(* IEC 61131-3 sources: PLC-Extruder-project/plc/twincat, 11 files *)

(* ---- DUT_ControllerState.st ---- *)
{attribute 'qualified_only'}
{attribute 'strict'}
TYPE E_ControllerState_Tc :
(
    IDLE := 0,
    STARTUP := 10,
    RUNNING := 20,
    SHUTDOWN := 30,
    EMERGENCY_STOP := 40
);
END_TYPE

(* ---- DUT_ExtruderApp.st ---- *)
{attribute 'qualified_only'}
{attribute 'strict'}
TYPE E_ExtruderMode_Tc :
(
    OFF := 0,
    MANUAL := 10,
    AUTO := 20,
    MAINTENANCE := 30
);
END_TYPE

{attribute 'qualified_only'}
{attribute 'strict'}
TYPE E_RecipeId_Tc :
(
    DEFAULT := 0,
    HDPE_PIPE := 10,
    PVC_PROFILE := 20,
    CUSTOM := 100
);
END_TYPE

TYPE ST_ExtruderRecipe :
STRUCT
    Name : STRING(32);
    Zone1Setpoint_C : LREAL;
    Zone2Setpoint_C : LREAL;
    Zone3Setpoint_C : LREAL;
    Zone4Setpoint_C : LREAL;
    DieSetpoint_C : LREAL;
    FeedRateKgH : LREAL;
    ScrewRpm : LREAL;
END_STRUCT
END_TYPE

TYPE ST_ExtruderPermissives :
STRUCT
    EStopHealthy : BOOL;
    GuardDoorClosed : BOOL;
    MotorDriveHealthy : BOOL;
    FeederDriveHealthy : BOOL;
    HopperMaterialAvailable : BOOL;
    ReadyToStart : BOOL;
END_STRUCT
END_TYPE

TYPE ST_ExtruderAlarmSummary :
STRUCT
    WarningCount : UINT;
    FaultCount : UINT;
    CriticalCount : UINT;
    AnyWarning : BOOL;
    AnyFault : BOOL;
    AnyCritical : BOOL;
    AlarmWord : DWORD;
END_STRUCT
END_TYPE

(* ---- DUT_ExtruderIo.st ---- *)
TYPE ST_ExtruderCommands :
STRUCT
    Start : BOOL;
    Stop : BOOL;
    Reset : BOOL;
    EmergencyStop : BOOL;
    Mode : E_ExtruderMode_Tc;
    RecipeId : E_RecipeId_Tc;
    RecipeFeedRateKgH : LREAL;
    RecipeScrewRpm : LREAL;
    Zone1Setpoint_C : LREAL;
    Zone2Setpoint_C : LREAL;
    Zone3Setpoint_C : LREAL;
    Zone4Setpoint_C : LREAL;
    DieSetpoint_C : LREAL;
END_STRUCT
END_TYPE

TYPE ST_ExtruderDigitalInputs :
STRUCT
    EStopOk : BOOL;
    GuardDoorClosed : BOOL;
    HeaterZone1Feedback : BOOL;
    HeaterZone2Feedback : BOOL;
    HeaterZone3Feedback : BOOL;
    HeaterZone4Feedback : BOOL;
    DieHeaterFeedback : BOOL;
    MotorDriveHealthy : BOOL;
    FeederDriveHealthy : BOOL;
END_STRUCT
END_TYPE

TYPE ST_ExtruderAnalogInputs :
STRUCT
    Zone1Temp_C : LREAL;
    Zone2Temp_C : LREAL;
    Zone3Temp_C : LREAL;
    Zone4Temp_C : LREAL;
    DieTemp_C : LREAL;
    MeltPressure_bar : LREAL;
    MotorRpm : LREAL;
    FeederRateKgH : LREAL;
    HopperLevelPct : LREAL;
    MotorCurrent_A : LREAL;
END_STRUCT
END_TYPE

TYPE ST_ExtruderDigitalOutputs :
STRUCT
    HeaterZone1Enable : BOOL;
    HeaterZone2Enable : BOOL;
    HeaterZone3Enable : BOOL;
    HeaterZone4Enable : BOOL;
    DieHeaterEnable : BOOL;
    MotorRunEnable : BOOL;
    FeederRunEnable : BOOL;
    StackLightRed : BOOL;
    StackLightAmber : BOOL;
    StackLightGreen : BOOL;
    Horn : BOOL;
END_STRUCT
END_TYPE

TYPE ST_ExtruderAnalogOutputs :
STRUCT
    HeaterZone1Pct : LREAL;
    HeaterZone2Pct : LREAL;
    HeaterZone3Pct : LREAL;
    HeaterZone4Pct : LREAL;
    DieHeaterPct : LREAL;
    MotorSpeedRefRpm : LREAL;
    FeederRateRefKgH : LREAL;
END_STRUCT
END_TYPE

TYPE ST_ExtruderStatus :
STRUCT
    State : E_ControllerState_Tc;
    SafetyState : E_SafetyState_Tc;
    Mode : E_ExtruderMode_Tc;
    ActiveRecipeId : E_RecipeId_Tc;
    ActiveRecipeName : STRING(32);
    ReadyToStart : BOOL;
    Running : BOOL;
    Faulted : BOOL;
    RunTime_s : LREAL;
    ScanNumber : UDINT;
    AnyWarning : BOOL;
    AnyAlarm : BOOL;
    HeaterAllAtSetpoint : BOOL;
    DieAtSetpoint : BOOL;
    FeedRateSetpointKgH : LREAL;
    ScrewRpmSetpoint : LREAL;
    Zone1Setpoint_C : LREAL;
    Zone2Setpoint_C : LREAL;
    Zone3Setpoint_C : LREAL;
    Zone4Setpoint_C : LREAL;
    DieSetpoint_C : LREAL;
    AlarmSummary : ST_ExtruderAlarmSummary;
    Permissives : ST_ExtruderPermissives;
END_STRUCT
END_TYPE

(* ---- DUT_SafetyState.st ---- *)
{attribute 'qualified_only'}
{attribute 'strict'}
TYPE E_SafetyState_Tc :
(
    SAFE := 0,
    WARNING := 10,
    E_STOP := 20
);
END_TYPE

(* ---- GVL_ExtruderConfig.st ---- *)
{attribute 'qualified_only'}
VAR_GLOBAL CONSTANT
    cCycleTime_s : LREAL := 0.1;

    cBarrelZone1Setpoint_C : LREAL := 180.0;
    cBarrelZone2Setpoint_C : LREAL := 200.0;
    cBarrelZone3Setpoint_C : LREAL := 220.0;
    cBarrelZone4Setpoint_C : LREAL := 230.0;
    cDieSetpoint_C : LREAL := 235.0;
    cTempTolerance_C : LREAL := 5.0;

    cMotorMinRpm : LREAL := 5.0;
    cMotorMaxRpm : LREAL := 150.0;
    cFeedMinKgH : LREAL := 5.0;
    cFeedMaxKgH : LREAL := 100.0;

    cDiePressureWarning_bar : LREAL := 300.0;
    cDiePressureMax_bar : LREAL := 350.0;
    cMaxBarrelTemp_C : LREAL := 280.0;

    cLowMaterialLevel_pct : LREAL := 10.0;
    cEmptyMaterialLevel_pct : LREAL := 2.0;
END_VAR

(* ---- GVL_ExtruderIo.st ---- *)
VAR_GLOBAL
    gExtruderCmd : ST_ExtruderCommands := (
        Mode := E_ExtruderMode_Tc.AUTO,
        RecipeId := E_RecipeId_Tc.DEFAULT,
        RecipeFeedRateKgH := 50.0,
        RecipeScrewRpm := 80.0,
        Zone1Setpoint_C := 180.0,
        Zone2Setpoint_C := 200.0,
        Zone3Setpoint_C := 220.0,
        Zone4Setpoint_C := 230.0,
        DieSetpoint_C := 235.0
    );

    gExtruderDI : ST_ExtruderDigitalInputs;
    gExtruderAI : ST_ExtruderAnalogInputs;

    gExtruderDO : ST_ExtruderDigitalOutputs;
    gExtruderAO : ST_ExtruderAnalogOutputs;

    gExtruderStatus : ST_ExtruderStatus := (
        State := E_ControllerState_Tc.IDLE,
        SafetyState := E_SafetyState_Tc.SAFE,
        Mode := E_ExtruderMode_Tc.AUTO,
        ActiveRecipeId := E_RecipeId_Tc.DEFAULT
    );
END_VAR

(* ---- GVL_ExtruderRecipes.st ---- *)
VAR_GLOBAL CONSTANT
    gcRecipeDefault : ST_ExtruderRecipe := (
        Name := 'Default Extrusion',
        Zone1Setpoint_C := 180.0,
        Zone2Setpoint_C := 200.0,
        Zone3Setpoint_C := 220.0,
        Zone4Setpoint_C := 230.0,
        DieSetpoint_C := 235.0,
        FeedRateKgH := 50.0,
        ScrewRpm := 80.0
    );

    gcRecipeHdpePipe : ST_ExtruderRecipe := (
        Name := 'HDPE Pipe',
        Zone1Setpoint_C := 175.0,
        Zone2Setpoint_C := 195.0,
        Zone3Setpoint_C := 210.0,
        Zone4Setpoint_C := 220.0,
        DieSetpoint_C := 225.0,
        FeedRateKgH := 62.0,
        ScrewRpm := 92.0
    );

    gcRecipePvcProfile : ST_ExtruderRecipe := (
        Name := 'PVC Profile',
        Zone1Setpoint_C := 165.0,
        Zone2Setpoint_C := 178.0,
        Zone3Setpoint_C := 186.0,
        Zone4Setpoint_C := 192.0,
        DieSetpoint_C := 195.0,
        FeedRateKgH := 42.0,
        ScrewRpm := 58.0
    );
END_VAR

(* ---- FB_AlarmManager_Tc.st ---- *)
FUNCTION_BLOCK FB_AlarmManager_Tc
VAR_INPUT
    Warning01 : BOOL;
    Warning02 : BOOL;
    Warning03 : BOOL;
    Warning04 : BOOL;
    Warning05 : BOOL;
    Fault01 : BOOL;
    Fault02 : BOOL;
    Fault03 : BOOL;
    Fault04 : BOOL;
    Critical01 : BOOL;
    Critical02 : BOOL;
    Critical03 : BOOL;
END_VAR
VAR_OUTPUT
    Summary : ST_ExtruderAlarmSummary;
END_VAR
VAR
    AlarmWord : DWORD;
END_VAR

Summary.WarningCount := 0;
Summary.FaultCount := 0;
Summary.CriticalCount := 0;
AlarmWord := DWORD#0;

IF Warning01 THEN Summary.WarningCount := Summary.WarningCount + 1; AlarmWord := AlarmWord OR DWORD#16#0001; END_IF;
IF Warning02 THEN Summary.WarningCount := Summary.WarningCount + 1; AlarmWord := AlarmWord OR DWORD#16#0002; END_IF;
IF Warning03 THEN Summary.WarningCount := Summary.WarningCount + 1; AlarmWord := AlarmWord OR DWORD#16#0004; END_IF;
IF Warning04 THEN Summary.WarningCount := Summary.WarningCount + 1; AlarmWord := AlarmWord OR DWORD#16#0008; END_IF;
IF Warning05 THEN Summary.WarningCount := Summary.WarningCount + 1; AlarmWord := AlarmWord OR DWORD#16#0010; END_IF;

IF Fault01 THEN Summary.FaultCount := Summary.FaultCount + 1; AlarmWord := AlarmWord OR DWORD#16#0100; END_IF;
IF Fault02 THEN Summary.FaultCount := Summary.FaultCount + 1; AlarmWord := AlarmWord OR DWORD#16#0200; END_IF;
IF Fault03 THEN Summary.FaultCount := Summary.FaultCount + 1; AlarmWord := AlarmWord OR DWORD#16#0400; END_IF;
IF Fault04 THEN Summary.FaultCount := Summary.FaultCount + 1; AlarmWord := AlarmWord OR DWORD#16#0800; END_IF;

IF Critical01 THEN Summary.CriticalCount := Summary.CriticalCount + 1; AlarmWord := AlarmWord OR DWORD#16#10000; END_IF;
IF Critical02 THEN Summary.CriticalCount := Summary.CriticalCount + 1; AlarmWord := AlarmWord OR DWORD#16#20000; END_IF;
IF Critical03 THEN Summary.CriticalCount := Summary.CriticalCount + 1; AlarmWord := AlarmWord OR DWORD#16#40000; END_IF;

Summary.AnyWarning := Summary.WarningCount > 0;
Summary.AnyFault := Summary.FaultCount > 0;
Summary.AnyCritical := Summary.CriticalCount > 0;
Summary.AlarmWord := AlarmWord;

END_FUNCTION_BLOCK

(* ---- FB_ExtruderController_Tc.st ---- *)
(*
    Beckhoff TwinCAT-oriented controller sequencer.

    TwinCAT details:
    - uses LREAL/UDINT
    - uses Standard library R_TRIG instances for edge detection
    - uses qualified enum names with strict typing
*)

FUNCTION_BLOCK FB_ExtruderController_Tc
VAR_INPUT
    StartCmd : BOOL;
    StopCmd : BOOL;
    ResetCmd : BOOL;
    EmergencyStopCmd : BOOL;

    SafetyEStop : BOOL;
    HeaterAllAtSetpoint : BOOL;
    DieAtSetpoint : BOOL;
    MotorActualRpm : LREAL;

    RecipeFeedRateCmd : LREAL := 50.0;
    RecipeScrewRpmCmd : LREAL := 80.0;
    FeedRateMin : LREAL := GVL_ExtruderConfig.cFeedMinKgH;
    FeedRateMax : LREAL := GVL_ExtruderConfig.cFeedMaxKgH;
    ScrewRpmMin : LREAL := GVL_ExtruderConfig.cMotorMinRpm;
    ScrewRpmMax : LREAL := GVL_ExtruderConfig.cMotorMaxRpm;
    CycleTime_s : LREAL := GVL_ExtruderConfig.cCycleTime_s;
END_VAR
VAR_OUTPUT
    State : E_ControllerState_Tc := E_ControllerState_Tc.IDLE;
    ScanNumber : UDINT := 0;
    RunTime_s : LREAL := 0.0;

    FeedRateSetpoint : LREAL := GVL_ExtruderConfig.cFeedMinKgH;
    ScrewRpmSetpoint : LREAL := GVL_ExtruderConfig.cMotorMinRpm;

    HeaterEnableCmd : BOOL := FALSE;
    DieEnableCmd : BOOL := FALSE;
    FeederRunCmd : BOOL := FALSE;
    MotorRunCmd : BOOL := FALSE;

    ResetSafetyCmd : BOOL := FALSE;
    ResetMotorFaultCmd : BOOL := FALSE;
    ResetFeederFaultCmd : BOOL := FALSE;

    RaiseShutdownAlarmCmd : BOOL := FALSE;
    ClearShutdownAlarmCmd : BOOL := FALSE;
    RaiseEStopAlarmCmd : BOOL := FALSE;
END_VAR
VAR
    PrevState : E_ControllerState_Tc := E_ControllerState_Tc.IDLE;
    rtStart : R_TRIG;
    rtStop : R_TRIG;
    rtReset : R_TRIG;
    rtEmergency : R_TRIG;
END_VAR

rtStart(CLK := StartCmd);
rtStop(CLK := StopCmd);
rtReset(CLK := ResetCmd);
rtEmergency(CLK := EmergencyStopCmd);

ResetSafetyCmd := FALSE;
ResetMotorFaultCmd := FALSE;
ResetFeederFaultCmd := FALSE;
RaiseShutdownAlarmCmd := FALSE;
ClearShutdownAlarmCmd := FALSE;
RaiseEStopAlarmCmd := FALSE;

ScanNumber := ScanNumber + 1;

FeedRateSetpoint := MAX(FeedRateMin, MIN(RecipeFeedRateCmd, FeedRateMax));
ScrewRpmSetpoint := MAX(ScrewRpmMin, MIN(RecipeScrewRpmCmd, ScrewRpmMax));

IF ((SafetyEStop OR rtEmergency.Q) AND
    (State <> E_ControllerState_Tc.EMERGENCY_STOP) AND
    (State <> E_ControllerState_Tc.IDLE)) THEN
    State := E_ControllerState_Tc.EMERGENCY_STOP;
END_IF;

CASE State OF
    E_ControllerState_Tc.IDLE:
        IF rtStart.Q THEN
            RunTime_s := 0.0;
            State := E_ControllerState_Tc.STARTUP;
        ELSIF rtReset.Q THEN
            RunTime_s := 0.0;
            ResetSafetyCmd := TRUE;
            ResetMotorFaultCmd := TRUE;
            ResetFeederFaultCmd := TRUE;
        END_IF;

    E_ControllerState_Tc.STARTUP:
        IF rtStop.Q THEN
            State := E_ControllerState_Tc.SHUTDOWN;
        ELSIF HeaterAllAtSetpoint AND DieAtSetpoint THEN
            State := E_ControllerState_Tc.RUNNING;
        END_IF;

    E_ControllerState_Tc.RUNNING:
        IF rtStop.Q THEN
            State := E_ControllerState_Tc.SHUTDOWN;
        ELSIF SafetyEStop OR rtEmergency.Q THEN
            State := E_ControllerState_Tc.EMERGENCY_STOP;
        ELSE
            RunTime_s := RunTime_s + CycleTime_s;
        END_IF;

    E_ControllerState_Tc.SHUTDOWN:
        IF SafetyEStop OR rtEmergency.Q THEN
            State := E_ControllerState_Tc.EMERGENCY_STOP;
        ELSIF MotorActualRpm < 0.5 THEN
            State := E_ControllerState_Tc.IDLE;
            ClearShutdownAlarmCmd := TRUE;
        END_IF;

    E_ControllerState_Tc.EMERGENCY_STOP:
        IF rtReset.Q THEN
            RunTime_s := 0.0;
            ResetSafetyCmd := TRUE;
            ResetMotorFaultCmd := TRUE;
            ResetFeederFaultCmd := TRUE;
            ClearShutdownAlarmCmd := TRUE;
            State := E_ControllerState_Tc.IDLE;
        END_IF;
END_CASE;

IF State <> PrevState THEN
    CASE State OF
        E_ControllerState_Tc.STARTUP:
            RunTime_s := 0.0;

        E_ControllerState_Tc.SHUTDOWN:
            RaiseShutdownAlarmCmd := TRUE;

        E_ControllerState_Tc.EMERGENCY_STOP:
            RaiseEStopAlarmCmd := TRUE;
    END_CASE;

    PrevState := State;
END_IF;

HeaterEnableCmd := (State = E_ControllerState_Tc.STARTUP) OR
                   (State = E_ControllerState_Tc.RUNNING) OR
                   (State = E_ControllerState_Tc.SHUTDOWN);
DieEnableCmd := HeaterEnableCmd;
FeederRunCmd := (State = E_ControllerState_Tc.RUNNING);
MotorRunCmd := (State = E_ControllerState_Tc.RUNNING);

END_FUNCTION_BLOCK

(* ---- FB_RecipeManager_Tc.st ---- *)
FUNCTION_BLOCK FB_RecipeManager_Tc
VAR_INPUT
    SelectedRecipeId : E_RecipeId_Tc;
    CustomRecipe : ST_ExtruderRecipe;
END_VAR
VAR_OUTPUT
    ActiveRecipeId : E_RecipeId_Tc := E_RecipeId_Tc.DEFAULT;
    ActiveRecipe : ST_ExtruderRecipe;
END_VAR

CASE SelectedRecipeId OF
    E_RecipeId_Tc.HDPE_PIPE:
        ActiveRecipeId := E_RecipeId_Tc.HDPE_PIPE;
        ActiveRecipe := GVL_ExtruderRecipes.gcRecipeHdpePipe;

    E_RecipeId_Tc.PVC_PROFILE:
        ActiveRecipeId := E_RecipeId_Tc.PVC_PROFILE;
        ActiveRecipe := GVL_ExtruderRecipes.gcRecipePvcProfile;

    E_RecipeId_Tc.CUSTOM:
        ActiveRecipeId := E_RecipeId_Tc.CUSTOM;
        ActiveRecipe := CustomRecipe;

ELSE
    ActiveRecipeId := E_RecipeId_Tc.DEFAULT;
    ActiveRecipe := GVL_ExtruderRecipes.gcRecipeDefault;
END_CASE;

END_FUNCTION_BLOCK

(* ---- PRG_ExtruderCell_Tc.st ---- *)
(*
    Beckhoff TwinCAT integration example for the extruder cell.

    Notes:
    - Map *_PV variables to EtherCAT or terminal I/O.
    - For production work, replace the generic component blocks with
      TwinCAT library-backed FBs where appropriate.
*)

PROGRAM PRG_ExtruderCell_Tc
VAR
    Ctrl : FB_ExtruderController_Tc;
    RecipeMgr : FB_RecipeManager_Tc;
    AlarmMgr : FB_AlarmManager_Tc;
    Zone1 : FB_HeatingZone;
    Zone2 : FB_HeatingZone;
    Zone3 : FB_HeatingZone;
    Zone4 : FB_HeatingZone;
    Die : FB_DieZone;
    Feeder : FB_MaterialFeeder;
    Motor : FB_ExtrusionMotor;
    ActiveRecipe : ST_ExtruderRecipe;
    CustomRecipe : ST_ExtruderRecipe;
    SafetyState : E_SafetyState_Tc := E_SafetyState_Tc.SAFE;
    SafetyEStopActive : BOOL;
    AnyWarning : BOOL;
    AnyFault : BOOL;
    AutoStartPermissive : BOOL;
    Permissives : ST_ExtruderPermissives;
END_VAR

CustomRecipe.Name := 'Custom';
CustomRecipe.Zone1Setpoint_C := gExtruderCmd.Zone1Setpoint_C;
CustomRecipe.Zone2Setpoint_C := gExtruderCmd.Zone2Setpoint_C;
CustomRecipe.Zone3Setpoint_C := gExtruderCmd.Zone3Setpoint_C;
CustomRecipe.Zone4Setpoint_C := gExtruderCmd.Zone4Setpoint_C;
CustomRecipe.DieSetpoint_C := gExtruderCmd.DieSetpoint_C;
CustomRecipe.FeedRateKgH := gExtruderCmd.RecipeFeedRateKgH;
CustomRecipe.ScrewRpm := gExtruderCmd.RecipeScrewRpm;

RecipeMgr(
    SelectedRecipeId := gExtruderCmd.RecipeId,
    CustomRecipe := CustomRecipe
);
ActiveRecipe := RecipeMgr.ActiveRecipe;

Permissives.EStopHealthy := gExtruderDI.EStopOk;
Permissives.GuardDoorClosed := gExtruderDI.GuardDoorClosed;
Permissives.MotorDriveHealthy := gExtruderDI.MotorDriveHealthy;
Permissives.FeederDriveHealthy := gExtruderDI.FeederDriveHealthy;
Permissives.HopperMaterialAvailable := gExtruderAI.HopperLevelPct > GVL_ExtruderConfig.cEmptyMaterialLevel_pct;
Permissives.ReadyToStart :=
    Permissives.EStopHealthy AND
    Permissives.GuardDoorClosed AND
    Permissives.MotorDriveHealthy AND
    Permissives.FeederDriveHealthy AND
    Permissives.HopperMaterialAvailable;

AutoStartPermissive :=
    (gExtruderCmd.Mode = E_ExtruderMode_Tc.AUTO) AND
    Permissives.ReadyToStart;

Zone1(
    EnableCmd := Ctrl.HeaterEnableCmd,
    ResetCmd := Ctrl.ResetSafetyCmd,
    TemperaturePV := REAL(gExtruderAI.Zone1Temp_C),
    Setpoint := REAL(ActiveRecipe.Zone1Setpoint_C),
    TempTolerance := REAL(GVL_ExtruderConfig.cTempTolerance_C),
    MaxTemp := REAL(GVL_ExtruderConfig.cMaxBarrelTemp_C)
);
Zone2(
    EnableCmd := Ctrl.HeaterEnableCmd,
    ResetCmd := Ctrl.ResetSafetyCmd,
    TemperaturePV := REAL(gExtruderAI.Zone2Temp_C),
    Setpoint := REAL(ActiveRecipe.Zone2Setpoint_C),
    TempTolerance := REAL(GVL_ExtruderConfig.cTempTolerance_C),
    MaxTemp := REAL(GVL_ExtruderConfig.cMaxBarrelTemp_C)
);
Zone3(
    EnableCmd := Ctrl.HeaterEnableCmd,
    ResetCmd := Ctrl.ResetSafetyCmd,
    TemperaturePV := REAL(gExtruderAI.Zone3Temp_C),
    Setpoint := REAL(ActiveRecipe.Zone3Setpoint_C),
    TempTolerance := REAL(GVL_ExtruderConfig.cTempTolerance_C),
    MaxTemp := REAL(GVL_ExtruderConfig.cMaxBarrelTemp_C)
);
Zone4(
    EnableCmd := Ctrl.HeaterEnableCmd,
    ResetCmd := Ctrl.ResetSafetyCmd,
    TemperaturePV := REAL(gExtruderAI.Zone4Temp_C),
    Setpoint := REAL(ActiveRecipe.Zone4Setpoint_C),
    TempTolerance := REAL(GVL_ExtruderConfig.cTempTolerance_C),
    MaxTemp := REAL(GVL_ExtruderConfig.cMaxBarrelTemp_C)
);

Feeder(
    RunCmd := Ctrl.FeederRunCmd,
    ResetCmd := Ctrl.ResetFeederFaultCmd,
    FeedRateSetpointKgH := REAL(Ctrl.FeedRateSetpoint),
    ActualRatePVKgH := REAL(gExtruderAI.FeederRateKgH),
    HopperLevelPctPV := REAL(gExtruderAI.HopperLevelPct),
    MinRateKgH := REAL(GVL_ExtruderConfig.cFeedMinKgH),
    MaxRateKgH := REAL(GVL_ExtruderConfig.cFeedMaxKgH),
    LowLevelPct := REAL(GVL_ExtruderConfig.cLowMaterialLevel_pct),
    EmptyLevelPct := REAL(GVL_ExtruderConfig.cEmptyMaterialLevel_pct)
);

Die(
    EnableCmd := Ctrl.DieEnableCmd,
    ResetCmd := Ctrl.ResetSafetyCmd,
    TemperaturePV := REAL(gExtruderAI.DieTemp_C),
    Setpoint := REAL(ActiveRecipe.DieSetpoint_C),
    TempTolerance := REAL(GVL_ExtruderConfig.cTempTolerance_C),
    MaxTemp := REAL(GVL_ExtruderConfig.cMaxBarrelTemp_C),
    ScrewRpmPV := REAL(gExtruderAI.MotorRpm),
    FeedRateActualKgH := REAL(gExtruderAI.FeederRateKgH),
    MotorMaxRpm := REAL(GVL_ExtruderConfig.cMotorMaxRpm),
    DieMaxPressureBar := REAL(GVL_ExtruderConfig.cDiePressureMax_bar),
    DieWarningPressureBar := REAL(GVL_ExtruderConfig.cDiePressureWarning_bar)
);

Motor(
    RunCmd := Ctrl.MotorRunCmd,
    ResetCmd := Ctrl.ResetMotorFaultCmd,
    SpeedSetpointRpm := REAL(Ctrl.ScrewRpmSetpoint),
    ActualRpmPV := REAL(gExtruderAI.MotorRpm),
    MeltPressureBar := REAL(gExtruderAI.MeltPressure_bar),
    MinRpm := REAL(GVL_ExtruderConfig.cMotorMinRpm),
    MaxRpm := REAL(GVL_ExtruderConfig.cMotorMaxRpm),
    DieMaxPressureBar := REAL(GVL_ExtruderConfig.cDiePressureMax_bar)
);

AnyWarning :=
    Zone1.UnderTempAlarm OR
    Zone2.UnderTempAlarm OR
    Zone3.UnderTempAlarm OR
    Zone4.UnderTempAlarm OR
    Die.HighPressureWarning OR
    Feeder.LowMaterialAlarm OR
    Motor.StallWarning;

AnyFault :=
    Feeder.FaultActive OR
    Motor.FaultActive;

SafetyEStopActive :=
    (NOT Permissives.EStopHealthy) OR
    (NOT Permissives.GuardDoorClosed) OR
    (NOT Permissives.MotorDriveHealthy) OR
    (NOT Permissives.FeederDriveHealthy) OR
    gExtruderCmd.EmergencyStop OR
    Zone1.OverTempAlarm OR
    Zone2.OverTempAlarm OR
    Zone3.OverTempAlarm OR
    Zone4.OverTempAlarm OR
    Die.OverPressureAlarm OR
    Motor.FaultActive;

AlarmMgr(
    Warning01 := Zone1.UnderTempAlarm,
    Warning02 := Zone2.UnderTempAlarm,
    Warning03 := Zone3.UnderTempAlarm,
    Warning04 := Zone4.UnderTempAlarm,
    Warning05 := Die.HighPressureWarning OR Feeder.LowMaterialAlarm OR Motor.StallWarning,
    Fault01 := Feeder.FaultActive,
    Fault02 := Motor.FaultActive,
    Fault03 := NOT Permissives.MotorDriveHealthy,
    Fault04 := NOT Permissives.FeederDriveHealthy,
    Critical01 := NOT Permissives.EStopHealthy OR gExtruderCmd.EmergencyStop,
    Critical02 := NOT Permissives.GuardDoorClosed,
    Critical03 := Zone1.OverTempAlarm OR Zone2.OverTempAlarm OR Zone3.OverTempAlarm OR Zone4.OverTempAlarm OR Die.OverPressureAlarm
);

IF SafetyEStopActive THEN
    SafetyState := E_SafetyState_Tc.E_STOP;
ELSIF AnyWarning THEN
    SafetyState := E_SafetyState_Tc.WARNING;
ELSE
    SafetyState := E_SafetyState_Tc.SAFE;
END_IF;

Ctrl(
    StartCmd := gExtruderCmd.Start AND AutoStartPermissive,
    StopCmd := gExtruderCmd.Stop OR (gExtruderCmd.Mode = E_ExtruderMode_Tc.OFF),
    ResetCmd := gExtruderCmd.Reset,
    EmergencyStopCmd := gExtruderCmd.EmergencyStop,
    SafetyEStop := SafetyEStopActive,
    HeaterAllAtSetpoint :=
        Zone1.AtSetpoint AND
        Zone2.AtSetpoint AND
        Zone3.AtSetpoint AND
        Zone4.AtSetpoint,
    DieAtSetpoint := Die.AtSetpoint,
    MotorActualRpm := gExtruderAI.MotorRpm,
    RecipeFeedRateCmd := ActiveRecipe.FeedRateKgH,
    RecipeScrewRpmCmd := ActiveRecipe.ScrewRpm,
    CycleTime_s := GVL_ExtruderConfig.cCycleTime_s
);

gExtruderDO.HeaterZone1Enable := Zone1.HeaterEnable;
gExtruderDO.HeaterZone2Enable := Zone2.HeaterEnable;
gExtruderDO.HeaterZone3Enable := Zone3.HeaterEnable;
gExtruderDO.HeaterZone4Enable := Zone4.HeaterEnable;
gExtruderDO.DieHeaterEnable := Die.HeaterEnable;
gExtruderDO.MotorRunEnable := Motor.MotorEnable;
gExtruderDO.FeederRunEnable := Feeder.FeederEnable;
gExtruderDO.StackLightRed := SafetyEStopActive;
gExtruderDO.StackLightAmber := AnyWarning AND NOT SafetyEStopActive;
gExtruderDO.StackLightGreen := Ctrl.State = E_ControllerState_Tc.RUNNING;
gExtruderDO.Horn := SafetyEStopActive;

gExtruderAO.HeaterZone1Pct := Zone1.HeaterOutputPct;
gExtruderAO.HeaterZone2Pct := Zone2.HeaterOutputPct;
gExtruderAO.HeaterZone3Pct := Zone3.HeaterOutputPct;
gExtruderAO.HeaterZone4Pct := Zone4.HeaterOutputPct;
gExtruderAO.DieHeaterPct := Die.HeaterOutputPct;
gExtruderAO.MotorSpeedRefRpm := Ctrl.ScrewRpmSetpoint;
gExtruderAO.FeederRateRefKgH := Ctrl.FeedRateSetpoint;

gExtruderStatus.State := Ctrl.State;
gExtruderStatus.SafetyState := SafetyState;
gExtruderStatus.Mode := gExtruderCmd.Mode;
gExtruderStatus.ActiveRecipeId := RecipeMgr.ActiveRecipeId;
gExtruderStatus.ActiveRecipeName := ActiveRecipe.Name;
gExtruderStatus.ReadyToStart := Permissives.ReadyToStart AND NOT SafetyEStopActive;
gExtruderStatus.Running := Ctrl.State = E_ControllerState_Tc.RUNNING;
gExtruderStatus.Faulted := SafetyEStopActive OR AnyFault;
gExtruderStatus.RunTime_s := Ctrl.RunTime_s;
gExtruderStatus.ScanNumber := Ctrl.ScanNumber;
gExtruderStatus.AnyWarning := AnyWarning;
gExtruderStatus.AnyAlarm := AlarmMgr.Summary.AnyWarning OR AlarmMgr.Summary.AnyFault OR AlarmMgr.Summary.AnyCritical;
gExtruderStatus.HeaterAllAtSetpoint :=
    Zone1.AtSetpoint AND
    Zone2.AtSetpoint AND
    Zone3.AtSetpoint AND
    Zone4.AtSetpoint;
gExtruderStatus.DieAtSetpoint := Die.AtSetpoint;
gExtruderStatus.FeedRateSetpointKgH := Ctrl.FeedRateSetpoint;
gExtruderStatus.ScrewRpmSetpoint := Ctrl.ScrewRpmSetpoint;
gExtruderStatus.Zone1Setpoint_C := ActiveRecipe.Zone1Setpoint_C;
gExtruderStatus.Zone2Setpoint_C := ActiveRecipe.Zone2Setpoint_C;
gExtruderStatus.Zone3Setpoint_C := ActiveRecipe.Zone3Setpoint_C;
gExtruderStatus.Zone4Setpoint_C := ActiveRecipe.Zone4Setpoint_C;
gExtruderStatus.DieSetpoint_C := ActiveRecipe.DieSetpoint_C;
gExtruderStatus.AlarmSummary := AlarmMgr.Summary;
gExtruderStatus.Permissives := Permissives;

END_PROGRAM
